Universal Robots PolyScope program: realtime_control.urp

Program realtime_control (installation=default directory=/ursim/programs createdIn=5.24.0 lastSavedIn=5.24.0 robotSerialNumber=20195599999)
Calibrated DH parameters: a=[0, -0.425, -0.3922, 0, 0, 0]; d=[0.1625, 0, 0, 0.1333, 0.0997, 0.0996]; alpha=[1.570796, 0, 0, 1.570796, -1.570796, 0]; deltaTheta=[0, 0, 0, 0, 0, 0]
InitVariablesNode
Robot Program (runOnlyOnce=false)
  Loop Forever
    new_pos := p[read_input_float_register(0),read_input_float_register(1),read_input_float_register(2),read_input_float_register(3),read_input_float_register(4),read_input_float_register(5)]
    If new_pos != p[0,0,0,0,0,0]
      Script: servoj(get_inverse_kin(new_pos), t=0.008, lookahead_time=0.1, gain=300)
    Script: sync()
